// TIA Portal V17 export
// export: Created 2022-12-08T07:31:25.9714192Z, ExportSetting WithDefaults, DisplayName Totally Integrated Automation Portal, DisplayVersion V17 Update 5, DisplayName TIA Portal Openness, DisplayVersion V17 Update 5, DisplayName TIA Portal Version Control Interface, DisplayVersion V17, DisplayName Simotion SCOUT TIA, DisplayVersion 5.4.3.0, DisplayName SINAMICS Startdrive Advanced, DisplayVersion V17 SP1, DisplayName SINAMICS Startdrive G130, G150, S120, S150, SINAMICS MV, S210, DisplayVersion V17 SP1, DisplayName SINAMICS Startdrive G110M, G120, G120C, G120D, G120P, G115D, DisplayVersion V17 SP1, DisplayName STEP 7 Professional, DisplayVersion V17 Update 5, DisplayName STEP 7 Safety, DisplayVersion V17, DisplayName WinCC Advanced, DisplayVersion V17 Update 5
DATA_BLOCK "BDE"   // DB710
{ S7_Optimized_Access := 'TRUE' }
AUTHOR : EconoPak GmbH
VERSION : 0.1
// stored: AutoNumber true, DBAccessibleFromOPCUA true, DBAccessibleFromWebserver true, InstanceOfName UDT_BDE, InstanceOfType UDT, IsOnlyStoredInLoadMemory false, IsWriteProtectedInAS false
"UDT_BDE"
   // VAR
   //    FaultCodeInformationMessages : Int;
   //    FaultCodeOperateMessages : Int;
   //    FaultCodeFaultMessagesAbsolut : Int;
   //    FaultCodeFaultMessagesCycleEnd : Int;
   //    ActualOMACMode : DInt;
   //    ActualOMACStatus : DInt;
   //    ProductCountOK : DInt;
   //    ProductCountNOK : DInt;
   //    ProductCountGesamt : DInt;
   // END_VAR
BEGIN
END_DATA_BLOCK
